(* IEC 61131-3 sources: pandora/pandora/aws-platform-main/aws-platform-main/src, 3 files *)

(* ---- AssetIdentifiers.st ---- *)
NAMESPACE Esab

    TYPE
        /// A complete list of possible assets
        AssetIdentifier : INT (
            Invalid := -1,

            GlobalState := 1,
            EmergencyStopCircuit := 2,
            Ups := 3,
            WeldSystemOrchestrator := 5,
            PowerSource1 := 6,
            PowerSource2 := 7,
            PowerSource3 := 8,
            FluxSystem := 10,
            RollerBed := 20,
            WeldHeadManipulator := 30,
            HorizontalSlideAxis := 31,
            VerticalSlideAxis := 32,

            PointLaser := 33,

            // P-HMI
            P_PushButton_EmergencyStop_Reset := 40,
            P_PushButton_FluxSystem_Release := 41,
            P_PushButton_FluxSystem_Recover := 42,
            P_PushButton_System_HighSpeed := 43,
            P_TwinPushButton_WireFeed1 := 44,
            P_TwinPushButton_WireFeed2 := 45,
            P_PushButton_MotionJoystick_AxisSelection := 46,
            P_Joystick_MotionJoystick := 47,
            P_PushButton_AxisJog_AxisSelection := 48,
            P_TwinPushButton_AxisJog := 49,
            P_PushButton_Start := 50,
            P_PushButton_Stop := 51,

            // C-HMI
            C_PushButton_EmergencyStop_Reset := 55,
            C_PushButton_FluxSystem_Release := 56,
            C_PushButton_System_HighSpeed := 57,
            C_TwinPushButton_WireFeed1 := 58,
            C_TwinPushButton_WireFeed2 := 59,
            C_TwinPushButton_WireFeed3 := 60,
            C_PushButton_TrackingOff := 61,
            C_Joystick_MotionJoystick := 62,
            C_TwinPushButton_Tilt := 63
        ) := AssetIdentifier#Invalid;
    END_TYPE

END_NAMESPACE

(* ---- GlobalState.st ---- *)
USING Esab.Utils.Alarming;
USING Esab.WeldSystem.Flux;
USING Esab.Motion;
USING Esab.Utils.Assets;
USING Esab.WeldSystem.PowerSources;

NAMESPACE Esab

    INTERFACE IGlobalState
        METHOD SetHighSpeed
            VAR_INPUT
                highSpeed : BOOL;
            END_VAR
        END_METHOD

        METHOD GetHighSpeed : BOOL
        END_METHOD

        METHOD SetMode
            VAR_INPUT
                mode : AwsPlatformMode;
            END_VAR
        END_METHOD

        METHOD GetMode : AwsPlatformMode
        END_METHOD
    END_INTERFACE

    CLASS GlobalState EXTENDS Asset IMPLEMENTS IGlobalState
        VAR PRIVATE
            _assets : IAssetsManager;
            _observable : GlobalStateObservable;

            _highSpeed : BOOL;
            _mode : AwsPlatformMode;

            _rollerBedObservable : REF_TO AxisObservable := NULL;
            _powerSource1Observable : REF_TO PowerSourceObservable := NULL;
            _powerSource2Observable : REF_TO PowerSourceObservable := NULL;
            _fluxSystemObservable : REF_TO FluxSystemObservable := NULL;
            _horizontalSlideAxisObservable : REF_TO AxisObservable := NULL;
            _verticalSlideAxisObservable : REF_TO AxisObservable := NULL;
        END_VAR

        METHOD PUBLIC Setup
            VAR_INPUT
                assets : IAssetsManager;
                setupAlarm : IAlarm;
            END_VAR

            _assets := assets;
            _setupAlarm := setupAlarm;

            _isSetup := _assets <> NULL;
        END_METHOD

        METHOD PUBLIC OVERRIDE Observe : IAssetObservable
            Observe := _observable;
        END_METHOD

        METHOD PUBLIC OVERRIDE Execute
            SUPER.Execute();

            IF _setupAlarm.IsActive() THEN
                RETURN;
            END_IF;
/*
            IF _rollerBedObservable = NULL THEN
                _rollerBedObservable ?= _assets.ObserveAsset(Esab.AssetIdentifier#RollerBed);
            END_IF;

            IF _powerSource1Observable = NULL THEN
                _powerSource1Observable ?= _assets.ObserveAsset(Esab.AssetIdentifier#PowerSource1);
            END_IF;

            IF _powerSource2Observable = NULL THEN
                _powerSource2Observable ?= _assets.ObserveAsset(Esab.AssetIdentifier#PowerSource2);
            END_IF;

            IF _fluxSystemObservable = NULL THEN
                _fluxSystemObservable ?= _assets.ObserveAsset(Esab.AssetIdentifier#FluxSystem);
            END_IF;

            IF _horizontalSlideAxisObservable = NULL THEN
                _horizontalSlideAxisObservable ?= _assets.ObserveAsset(Esab.AssetIdentifier#HorizontalSlideAxis);
            END_IF;

            IF _verticalSlideAxisObservable = NULL THEN
                _verticalSlideAxisObservable ?= _assets.ObserveAsset(Esab.AssetIdentifier#VerticalSlideAxis);
            END_IF;*/

            THIS.UpdateObservable();
        END_METHOD

        METHOD PUBLIC OVERRIDE UpdateState
            VAR_TEMP
                state : SystemState := SystemState#Healthy;
            END_VAR

            IF _rollerBedObservable <> NULL THEN
                IF _rollerBedObservable^.State = AxisState#Error THEN
                    state := SystemState#Error;
                END_IF;
            END_IF;

            IF _powerSource1Observable <> NULL THEN
                IF _powerSource1Observable^.State = PowerSourceState#Error THEN
                    state := SystemState#Error;
                END_IF;
            END_IF;

            IF _powerSource2Observable <> NULL THEN
                IF _powerSource2Observable^.State = PowerSourceState#Error THEN
                    state := SystemState#Error;
                END_IF;
            END_IF;

            IF _fluxSystemObservable <> NULL THEN
                IF _fluxSystemObservable^.State = FluxSystemState#Error THEN
                    state := SystemState#Error;
                END_IF;
            END_IF;

            IF _horizontalSlideAxisObservable <> NULL THEN
                IF _horizontalSlideAxisObservable^.Error THEN
                    state := SystemState#Error;
                END_IF;
            END_IF;

            IF _verticalSlideAxisObservable <> NULL THEN
                IF _verticalSlideAxisObservable^.Error THEN
                    state := SystemState#Error;
                END_IF;
            END_IF;

            _currentState := state;
        END_METHOD

        METHOD PUBLIC SetHighSpeed
            VAR_INPUT
                highSpeed : BOOL;
            END_VAR

            _highSpeed := highSpeed;
        END_METHOD

        METHOD PUBLIC GetHighSpeed : BOOL
            GetHighSpeed := _highSpeed;
        END_METHOD

        METHOD PUBLIC SetMode
            VAR_INPUT
                mode : AwsPlatformMode;
            END_VAR

            _mode := mode;
        END_METHOD

        METHOD PUBLIC GetMode : AwsPlatformMode
            GetMode := _mode;
        END_METHOD

        METHOD PRIVATE UpdateObservable
            _observable.HighSpeed := _highSpeed;
            _observable.Mode := _mode;
        END_METHOD
    END_CLASS

    CLASS GlobalStateObservable IMPLEMENTS IAssetObservable
        VAR PUBLIC
            State : SystemState;
            HighSpeed : BOOL := FALSE;
            Mode : AwsPlatformMode;
        END_VAR
    END_CLASS

    TYPE
        SystemState : INT(
            Healthy := 0,
            Error := 1
        );

        AwsPlatformMode : INT(
            Manual := 0,
            Adaptio := 1
        ) := AwsPlatformMode#Manual;
    END_TYPE

END_NAMESPACE

(* ---- Object.st ---- *)
USING Esab.Utils.Alarming;

USING Siemens.Simatic.S71500.Alarming;

NAMESPACE Esab

    CLASS Object
        VAR PROTECTED
            _isSetup : BOOL := FALSE;
            _setupAlarm : IAlarm := NULL;

            {S7.Alarm = NoAck, "Object not setup properly"}
            _defaultSetupAlarm : ProgramAlarm;
            _defaultSetupAlarmWrapper : AlarmWrapper;

            _currentState : INT;
        END_VAR

        METHOD PUBLIC Execute
            IF _setupAlarm = NULL THEN
                _defaultSetupAlarmWrapper.Setup(REF(_defaultSetupAlarm));
                _setupAlarm := _defaultSetupAlarmWrapper;
            END_IF;

            _setupAlarm.Execute(NOT _isSetup);

            THIS.UpdateState();
        END_METHOD

        /// Updates the current object status (state), by default it is set to 0 which should signify "OK/healthy/idle" in all implementers.
        METHOD PUBLIC UpdateState
            _currentState := 0;
        END_METHOD

        METHOD PUBLIC GetState : INT
            GetState := _currentState;
        END_METHOD
    END_CLASS

END_NAMESPACE
